Fanuc KAREL source: SET_PORT_ASG.kl

PROGRAM T
%NOLOCKGROUP
VAR
 v0 : INTEGER
 v1 : INTEGER
 v2 : INTEGER
 v3 : INTEGER
 v4 : INTEGER
 v5 : INTEGER
 v6 : INTEGER
 v7 : INTEGER
BEGIN
 SET_PORT_ASG(v0, v1, v2, v3, v4, v5, v6, v7)
END T
